(* IEC 61131-3 sources: Std_PalletMover/Class/AgvConfig, 1 file *)

(* ---- AgvConfig.st ---- *)
(*!
<Class
	Name               = "AgvConfig"
	Revision           = "0.0"
	RealtimeTask       = "false"
	CyclicTask         = "false"
	BackgroundTask     = "false"
	Sigmatek           = "false"
	OSInterface        = "false"
	HighPriority       = "false"
	Automatic          = "false"
	UpdateMode         = "Prescan"
	SharedCommandTable = "true"
	Objectsize         = "(690,240)">
	<Channels>
		<Server Name="Command" Visualized="false" Initialize="false" WriteProtected="false" Retentive="false"/>
	</Channels>
	<Network Name="AgvConfig">
		<!-- List of Components in this network -->
		<Components>
			<Object
				Name       = "_base"
				Class      = "_SettingsBase"
				Position   = "(218,120)"
				Visualized = "false">
				<Channels>
					<Server Name="ClassSvr"/>
					<Server Name="ItemError"/>
					<Server Name="ItemOk"/>
					<Client Name="op_LogData"/>
				</Channels>
			</Object>
		</Components>
		<Comments>
		</Comments>
		<!-- List of Connections in this network -->
		<Connections>
			<Connection Source="this.ClassSvr" Destination="_base.ClassSvr" Vertices="(826,210),(654,210),"/>
			<Connection Source="this.ItemOk" Destination="_base.ItemOk" Vertices="(826,270),(654,270),"/>
			<Connection Source="this.ItemError" Destination="_base.ItemError" Vertices="(826,330),(654,330),"/>
			<Connection Source="_base.op_LogData" Destination="this.op_LogData" Vertices="(218,210),(38,210),"/>
		</Connections>
		<!-- Headerfiles -->
		<Options>
		</Options>
	</Network>
</Class>
*)
#pragma using _Settingsbase

AgvConfig : CLASS
: _Settingsbase
  //Servers:
	Command 	: SvrCh_gt_AgvSettingsCmd;
  //Clients:
  //Variables:
  //Functions:

	FUNCTION VIRTUAL GLOBAL Init;

	FUNCTION VIRTUAL GLOBAL Command::Read
		VAR_OUTPUT
			output (EAX) 	: gt_AgvSettingsCmd;
		END_VAR;

	FUNCTION VIRTUAL GLOBAL Command::Write
		VAR_INPUT
			input (EAX) 	: gt_AgvSettingsCmd;
		END_VAR
		VAR_OUTPUT
			result (EAX) 	: gt_AgvSettingsCmd;
		END_VAR;
  //Tables:
	FUNCTION @STD
		VAR_OUTPUT
			ret_code	: CONFSTATES;
		END_VAR;
	FUNCTION GLOBAL TAB @CT_;
END_CLASS;

FUNCTION VIRTUAL GLOBAL AgvConfig::Command::Write
	VAR_INPUT
		input (EAX) 	: gt_AgvSettingsCmd;
	END_VAR
	VAR_OUTPUT
		result (EAX) 	: gt_AgvSettingsCmd;
	END_VAR

	Command := input;
    case  Command  of

        LoadSettings:

            if UpdateFile(Name:="c:\settings\machinesettings.json") = true then
    	        result := LoadLoading;
            else
                result:= LoadReadError;
            end_if;

            else

                   result:= LoadReadError;
      end_case;
       Command := result;
END_FUNCTION

FUNCTION VIRTUAL GLOBAL AgvConfig::Command::Read
	VAR_OUTPUT
		output (EAX) 	: gt_AgvSettingsCmd;
	END_VAR

    if JSreader.ReadFSM.Read() = _JSONReader::t_e_READSTEPS::RS_COMPLETE then
          pObjectHandle := JsReader.GetMainElement();
          if pObjectHandle <> nil then
              Command := ::gt_AgvSettingsCmd::LoadReadyOk;
           end_if;
    end_if;

	output := Command;

END_FUNCTION

FUNCTION VIRTUAL GLOBAL AgvConfig::Init

END_FUNCTION
